KUKA KRL program: p01drop_1711.src, p01drop_1711.dat

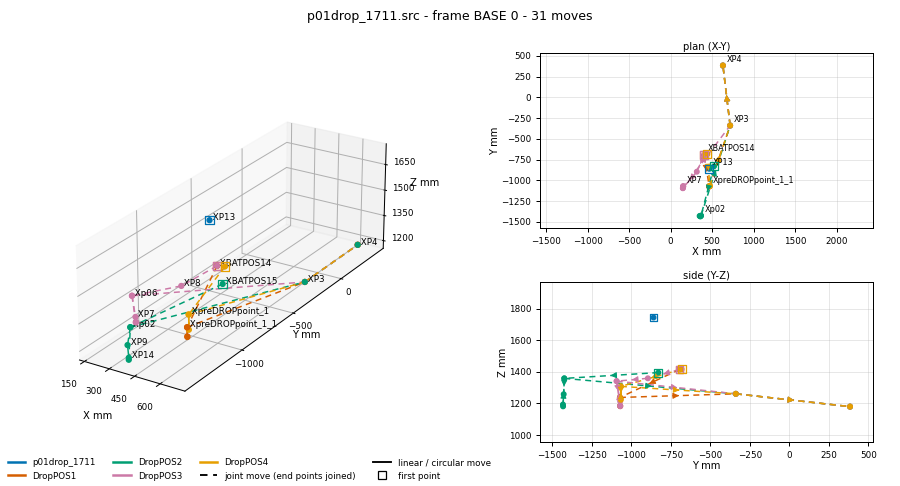
[picture p0: tool path of p01drop_1711.src in frame BASE 0, 31 of 34 moves have a stored position in this frame; points joined in program order, loops and branches not executed]
--- p01drop_1711.src ---
&ACCESS RVP1
&COMMENT Drop Part
&PARAM EDITMASK = *
&PARAM TEMPLATE = C:\KRC\Roboter\Template\vorgabe
&PARAM DISKPATH = KRC:\R1\Program\Sub Programs
DEF p01drop_1711( )
;FOLD INI
  ;FOLD BASISTECH INI

    GLOBAL INTERRUPT DECL 3 WHEN $STOPMESS==TRUE DO IR_STOPM ( )
    INTERRUPT ON 3
    BAS (#INITMOV,0 )
  ;ENDFOLD (BASISTECH INI)
;ENDFOLD (INI)
;================================================
; MODEL    : XXXX
; IE GROUP : XX
; STATION  : XXX
; ROBOT    : RX
; FUNCTION : Drop Part in StXX
;================================================
$TIMER[7]=0
$TIMER_STOP[7]=FALSE

waitarea:
QR_NOK=FALSE

;Wait For Area / Goto Safety / Return To Home

;FOLD PTP P13 Vel=100 % PDAT28 Tool[1] Base[0];%{PE}%R 8.3.48,%MKUKATPBASIS,%CMOVE,%VPTP,%P 1:PTP, 2:P13, 3:, 5:100, 7:PDAT28
$BWDSTART=FALSE
PDAT_ACT=PPDAT28
FDAT_ACT=FP13
BAS(#PTP_PARAMS,100)
PTP XP13
;ENDFOLD
;IF FALSE THEN


WAIT FOR ($IN[54]==TRUE) OR ($IN[1]==TRUE)

IF $in[54]==TRUE THEN
   bomberos_2 ( )               ; PICK In Station XX
   ENDIF


;Para de contar TC hasta que recibe typinfo para dejar (paleta indexada, tipo...)
$TIMER_STOP[7]=TRUE

;FOLD TYPE INFO

WAIT FOR ($IN[54]==TRUE) OR ($IN[1]==TRUE)
IF $in[54]==TRUE THEN
   bomberos_2 ( )               ; PICK In Station XX
   ENDIF
O_TYPE_REQ=FALSE
WAIT FOR I_TYPE_INFO==0
O_TYPE_REQ=TRUE
WAIT FOR ((I_TYPE_INFO>100) AND (I_TYPE_INFO<201) or ($IN[54]==TRUE))
IF $in[54]==TRUE THEN
   bomberos_2 ( )               ; PICK In Station XX
   ENDIF
O_TYPE_INFO=I_TYPE_INFO
;ENDFOLD
;ENDIF

$TIMER_STOP[7]=FALSE

SWITCH i_TYPE_INFO ;coldplate grande o peq


CASE 111
   INDICE_DROP=1 ;Variable calculo TC
   O_TYPE_REQ=FALSE
   DropPOS1() ;POSICION 1 COLDPLATE GRANDE

CASE 112
   INDICE_DROP=2  ;Variable calculo TC
   O_TYPE_REQ=FALSE
   DropPOS2() ;POSICION 2 COLDPLATE GRANDE

CASE 113
   INDICE_DROP=3
   O_TYPE_REQ=FALSE
   DropPOS3() ;POSICION 3 COLDPLATE GRANDE

CASE 121
   INDICE_DROP=4
   O_TYPE_REQ=FALSE
   DropPOS1();POSICION 1 COLDPLATE PEQUEÑO

CASE 200
   INDICE_DROP=4
   O_TYPE_REQ=FALSE
   P01DROP2_2();POSICION 1 COLDPLATE PEQUEÑO

CASE 155
   O_TYPE_REQ=FALSE
   bomberos_2() ;POSICION 1 COLDPLATE GRANDE
DEFAULT

WAIT FOR FALSE

ENDSWITCH

;fold QR NOK
IF (QR_NOK==TRUE) THEN

GOTO waitarea
ENDIF

;ENDFOLD


;FOLD PROVISIONAL PARA PRUEBAS
IF M2_TYPE_INFO<13 THEN
M2_TYPE_INFO=M2_TYPE_INFO+1
ENDIF

;ENDFOLD

PEXIT:

;FOLD Guarda_TC Dejada

;Guarda TC dejada
$TIMER_STOP[7]=TRUE
TC_DROP[INDICE_DROP]=$TIMER[7]

IF (INDICE_DROP < 4) THEN ;CUANDO DEJA ARRAYS EN COLD PLATES GRANDES
   IF (INDICE_RACK == 1)THEN
      TC_CP_BIG[INDICE_DROP]=TC_DROP[INDICE_DROP]+TC_PICK_RACK1[INDICE_PICK]
   ELSE
      TC_CP_BIG[INDICE_DROP]=TC_DROP[INDICE_DROP]+TC_PICK_RACK2[INDICE_PICK]
   ENDIF
   IF (INDICE_DROP == 3) THEN ;Cuando rellena el tercer colplate acumula en array de CP big
      TC_ARRAY_CPB[INDICE_ARRAYS_CPB]=TC_CP_BIG[1]+TC_CP_BIG[2]+TC_CP_BIG[3]
      INDICE_ARRAYS_CPB=INDICE_ARRAYS_CPB+1
      IF (INDICE_ARRAYS_CPB > 18) THEN
         INDICE_ARRAYS_CPB=1
         ;Actualiza el tiempo de ciclo medio por bateria
         ;Toma el tiempo de ciclo medio por batería como la media de procesar 2 racks
         ;64 arrays y 4 cartones, eso vienen a ser unas 7 baterías y me sobra 1 array
         TC_MEDIO_CARTONES=((((TC_CARTON[1]+TC_CARTON[2]+TC_CARTON[3]+TC_CARTON[4])/1000)*63)/64)
         TC_MEDIO_BATERIA=((TC_ARRAY_CPB[1]+TC_ARRAY_CPB[2]+TC_ARRAY_CPB[3]+TC_ARRAY_CPB[4]+TC_ARRAY_CPB[5]+TC_ARRAY_CPB[6]+TC_ARRAY_CPB[7]+TC_ARRAY_CPB[8]+TC_ARRAY_CPB[9]+TC_ARRAY_CPB[10]+TC_ARRAY_CPB[11]+TC_ARRAY_CPB[12]+TC_ARRAY_CPB[13]+TC_ARRAY_CPB[14]+TC_ARRAY_CPB[15]+TC_ARRAY_CPB[16]+TC_ARRAY_CPB[17]+TC_ARRAY_CPB[18]+TC_CP_SMALL[1]+TC_CP_SMALL[2]+TC_CP_SMALL[3]+TC_CP_SMALL[4]+TC_CP_SMALL[5]+TC_CP_SMALL[6]+TC_CP_SMALL[7]+TC_CP_SMALL[8]+TC_CP_SMALL[9])/1000)
         TC_MEDIO_BATERIA=((TC_MEDIO_BATERIA+TC_MEDIO_CARTONES)/9)
      ENDIF
   ENDIF
      ENDIF

IF (INDICE_DROP == 4) THEN ;CUANDO DEJA ARRAYS EN COLD PLATE PEQUEÑOS
   IF (INDICE_RACK == 1)THEN
      TC_CP_SMALL[INDICE_ARRAYS_CPS]=TC_DROP[4]+TC_PICK_RACK1[INDICE_PICK]
   ELSE
      TC_CP_SMALL[INDICE_ARRAYS_CPS]=TC_DROP[4]+TC_PICK_RACK2[INDICE_PICK]
   ENDIF
   INDICE_ARRAYS_CPS=INDICE_ARRAYS_CPS+1
   IF (INDICE_ARRAYS_CPS > 9) THEN
      INDICE_ARRAYS_CPS=1
   ENDIF
ENDIF

;ENDFOLD

END
DEF       DropPOS1()


;FOLD PTP BATPOS14 Vel=100 % PDAT9 Tool[8]:Gripper_array Base[0];%{PE}%R 8.3.48,%MKUKATPBASIS,%CMOVE,%VPTP,%P 1:PTP, 2:BATPOS14, 3:, 5:100, 7:PDAT9
$BWDSTART=FALSE
PDAT_ACT=PPDAT9
FDAT_ACT=FBATPOS14
BAS(#PTP_PARAMS,100)
PTP XBATPOS14
;ENDFOLD
;Wait For Area / Goto Safety / Return To Home

;FOLD Fordtech.Area_Req Area Request: 3, Safety Position: 0, Return To Home: 0 ;%{PE}
Area_Req (3,0,0)
IF I_RETHP AND (0 <> 0) AND ($IN_HOME == TRUE) THEN
  GOTO PEXIT
ENDIF
;ENDFOLD


;FOLD PTP preDROPpoint_1_1 CONT Vel=100 % PDAT9 Tool[8]:Gripper_array Base[0];%{PE}%R 8.3.48,%MKUKATPBASIS,%CMOVE,%VPTP,%P 1:PTP, 2:preDROPpoint_1_1, 3:C_DIS, 5:100, 7:PDAT9
$BWDSTART=FALSE
PDAT_ACT=PPDAT9
FDAT_ACT=FpreDROPpoint_1_1
BAS(#PTP_PARAMS,100)
PTP XpreDROPpoint_1_1 C_DIS
;ENDFOLD

;Pto antes de tocar TIM inclina vert
;FOLD LIN P11 Vel=2 m/s CPDAT9 Tool[8]:Gripper_array Base[0];%{PE}%R 8.3.48,%MKUKATPBASIS,%CMOVE,%VLIN,%P 1:LIN, 2:P11, 3:, 5:2, 7:CPDAT9
$BWDSTART=FALSE
LDAT_ACT=LCPDAT9
FDAT_ACT=FP11
BAS(#CP_PARAMS,2)
LIN XP11
;ENDFOLD
;FOLD WAIT Time=0.3 sec;%{PE}%R 8.3.48,%MKUKATPBASIS,%CWAIT,%VWAIT,%P 3:0.3
WAIT SEC 0.3
;ENDFOLD

;FOLD LIN DROPpoint_1_1 Vel=0.0025 m/s L2 Tool[8]:Gripper_array Base[0];%{PE}%R 8.3.48,%MKUKATPBASIS,%CMOVE,%VLIN,%P 1:LIN, 2:DROPpoint_1_1, 3:, 5:0.0025, 7:L2
$BWDSTART=FALSE
LDAT_ACT=LL2
FDAT_ACT=FDROPpoint_1_1
BAS(#CP_PARAMS,0.0025)
LIN XDROPpoint_1_1
;ENDFOLD

;abrir gara
cil_bat_reposo()

;FOLD PTP preDROPpoint_1_1 CONT Vel=100 % PDAT20 Tool[8]:Gripper_array Base[0];%{PE}%R 8.3.48,%MKUKATPBASIS,%CMOVE,%VPTP,%P 1:PTP, 2:preDROPpoint_1_1, 3:C_DIS, 5:100, 7:PDAT20
$BWDSTART=FALSE
PDAT_ACT=PPDAT20
FDAT_ACT=FpreDROPpoint_1_1
BAS(#PTP_PARAMS,100)
PTP XpreDROPpoint_1_1 C_DIS
;ENDFOLD
;FOLD SYN OUT 43 'Job Ready 3' State=TRUE at START Delay=0 ms;%{PE}%R 8.3.48,%MKUKATPBASIS,%COUT,%VSYNOUT,%P 2:43, 3:Job Ready 3, 5:TRUE, 7:0, 9:0, 12:0
TRIGGER WHEN DISTANCE=0 DELAY=0 DO $OUT[43]=TRUE
;ENDFOLD


;FOLD PTP P3 CONT Vel=100 % PDAT9 Tool[5] Base[0];%{PE}%R 8.3.48,%MKUKATPBASIS,%CMOVE,%VPTP,%P 1:PTP, 2:P3, 3:C_DIS, 5:100, 7:PDAT9
$BWDSTART=FALSE
PDAT_ACT=PPDAT9
FDAT_ACT=FP3
BAS(#PTP_PARAMS,100)
PTP XP3 C_DIS
;ENDFOLD

;Release Area 1
;FOLD SYN OUT 19 'Area Release 3' State=TRUE at START Delay=0 ms;%{PE}%R 8.3.48,%MKUKATPBASIS,%COUT,%VSYNOUT,%P 2:19, 3:Area Release 3, 5:TRUE, 7:0, 9:0, 12:0
TRIGGER WHEN DISTANCE=0 DELAY=0 DO $OUT[19]=TRUE
;ENDFOLD


;FOLD PTP P4 CONT Vel=100 % PDAT9 Tool[5] Base[0];%{PE}%R 8.3.48,%MKUKATPBASIS,%CMOVE,%VPTP,%P 1:PTP, 2:P4, 3:C_DIS, 5:100, 7:PDAT9
$BWDSTART=FALSE
PDAT_ACT=PPDAT9
FDAT_ACT=FP4
BAS(#PTP_PARAMS,100)
PTP XP4 C_DIS
;ENDFOLD

;FOLD PTP HOME Vel=100 % DEFAULT;%{PE}%R 8.3.48,%MKUKATPBASIS,%CMOVE,%VPTP,%P 1:PTP, 2:HOME, 3:, 5:100, 7:DEFAULT
$BWDSTART=FALSE
PDAT_ACT=PDEFAULT
FDAT_ACT=FHOME
BAS(#PTP_PARAMS,100)
$H_POS=XHOME
PTP XHOME
;ENDFOLD
;Jump Adress
PEXIT:



END

DEF       DropPOS2()

;FOLD PTP BATPOS15 Vel=100 % PDAT11 Tool[8]:Gripper_array Base[0];%{PE}%R 8.3.48,%MKUKATPBASIS,%CMOVE,%VPTP,%P 1:PTP, 2:BATPOS15, 3:, 5:100, 7:PDAT11
$BWDSTART=FALSE
PDAT_ACT=PPDAT11
FDAT_ACT=FBATPOS15
BAS(#PTP_PARAMS,100)
PTP XBATPOS15
;ENDFOLD
;Wait For Area / Goto Safety / Return To Home

;FOLD Fordtech.Area_Req Area Request: 3, Safety Position: 0, Return To Home: 0 ;%{PE}
Area_Req (3,0,0)
IF I_RETHP AND (0 <> 0) AND ($IN_HOME == TRUE) THEN
  GOTO PEXIT
ENDIF
;ENDFOLD

;predrop pos
;FOLD PTP p02 CONT Vel=100 % PDAT12 Tool[8]:Gripper_array Base[0];%{PE}%R 8.3.48,%MKUKATPBASIS,%CMOVE,%VPTP,%P 1:PTP, 2:p02, 3:C_DIS, 5:100, 7:PDAT12
$BWDSTART=FALSE
PDAT_ACT=PPDAT12
FDAT_ACT=Fp02
BAS(#PTP_PARAMS,100)
PTP Xp02 C_DIS
;ENDFOLD
;FOLD PTP P9 CONT Vel=100 % PDAT27 Tool[8]:Gripper_array Base[0];%{PE}%R 8.3.48,%MKUKATPBASIS,%CMOVE,%VPTP,%P 1:PTP, 2:P9, 3:C_DIS, 5:100, 7:PDAT27
$BWDSTART=FALSE
PDAT_ACT=PPDAT27
FDAT_ACT=FP9
BAS(#PTP_PARAMS,100)
PTP XP9 C_DIS
;ENDFOLD

;Pto antes de tocar TIM inclina hor
;FOLD LIN P14 Vel=2 m/s CPDAT12 Tool[8]:Gripper_array Base[0];%{PE}%R 8.3.48,%MKUKATPBASIS,%CMOVE,%VLIN,%P 1:LIN, 2:P14, 3:, 5:2, 7:CPDAT12
$BWDSTART=FALSE
LDAT_ACT=LCPDAT12
FDAT_ACT=FP14
BAS(#CP_PARAMS,2)
LIN XP14
;ENDFOLD
;FOLD WAIT Time=0.3 sec;%{PE}%R 8.3.48,%MKUKATPBASIS,%CWAIT,%VWAIT,%P 3:0.3
WAIT SEC 0.3
;ENDFOLD

;drop pos
;FOLD LIN p01 Vel=0.005 m/s L2 Tool[8]:Gripper_array Base[0];%{PE}%R 8.3.48,%MKUKATPBASIS,%CMOVE,%VLIN,%P 1:LIN, 2:p01, 3:, 5:0.005, 7:L2
$BWDSTART=FALSE
LDAT_ACT=LL2
FDAT_ACT=Fp01
BAS(#CP_PARAMS,0.005)
LIN Xp01
;ENDFOLD

;abrir gara
cil_bat_reposo()

;FOLD PTP p02 CONT Vel=100 % PDAT21 Tool[8]:Gripper_array Base[0];%{PE}%R 8.3.48,%MKUKATPBASIS,%CMOVE,%VPTP,%P 1:PTP, 2:p02, 3:C_DIS, 5:100, 7:PDAT21
$BWDSTART=FALSE
PDAT_ACT=PPDAT21
FDAT_ACT=Fp02
BAS(#PTP_PARAMS,100)
PTP Xp02 C_DIS
;ENDFOLD

;FOLD SYN OUT 43 'Job Ready 3' State=TRUE at START Delay=0 ms;%{PE}%R 8.3.48,%MKUKATPBASIS,%COUT,%VSYNOUT,%P 2:43, 3:Job Ready 3, 5:TRUE, 7:0, 9:0, 12:0
TRIGGER WHEN DISTANCE=0 DELAY=0 DO $OUT[43]=TRUE
;ENDFOLD

;FOLD PTP p03 CONT Vel=100 % PDAT13 Tool[5] Base[0];%{PE}%R 8.3.48,%MKUKATPBASIS,%CMOVE,%VPTP,%P 1:PTP, 2:p03, 3:C_DIS, 5:100, 7:PDAT13
$BWDSTART=FALSE
PDAT_ACT=PPDAT13
FDAT_ACT=Fp03
BAS(#PTP_PARAMS,100)
PTP Xp03 C_DIS
;ENDFOLD

;Release Area 1
;FOLD SYN OUT 19 'Area Release 3' State=TRUE at START Delay=0 ms;%{PE}%R 8.3.48,%MKUKATPBASIS,%COUT,%VSYNOUT,%P 2:19, 3:Area Release 3, 5:TRUE, 7:0, 9:0, 12:0
TRIGGER WHEN DISTANCE=0 DELAY=0 DO $OUT[19]=TRUE
;ENDFOLD


;FOLD PTP p04 CONT Vel=100 % PDAT14 Tool[5] Base[0];%{PE}%R 8.3.48,%MKUKATPBASIS,%CMOVE,%VPTP,%P 1:PTP, 2:p04, 3:C_DIS, 5:100, 7:PDAT14
$BWDSTART=FALSE
PDAT_ACT=PPDAT14
FDAT_ACT=Fp04
BAS(#PTP_PARAMS,100)
PTP Xp04 C_DIS
;ENDFOLD

;FOLD PTP HOME Vel=100 % DEFAULT;%{PE}%R 8.3.48,%MKUKATPBASIS,%CMOVE,%VPTP,%P 1:PTP, 2:HOME, 3:, 5:100, 7:DEFAULT
$BWDSTART=FALSE
PDAT_ACT=PDEFAULT
FDAT_ACT=FHOME
BAS(#PTP_PARAMS,100)
$H_POS=XHOME
PTP XHOME
;ENDFOLD
;Jump Adress
PEXIT:

END
DEF       DropPOS3()

;FOLD PTP BATPOS16 Vel=100 % PDAT17 Tool[8]:Gripper_array Base[0];%{PE}%R 8.3.48,%MKUKATPBASIS,%CMOVE,%VPTP,%P 1:PTP, 2:BATPOS16, 3:, 5:100, 7:PDAT17
$BWDSTART=FALSE
PDAT_ACT=PPDAT17
FDAT_ACT=FBATPOS16
BAS(#PTP_PARAMS,100)
PTP XBATPOS16
;ENDFOLD
;Wait For Area / Goto Safety / Return To Home

;FOLD Fordtech.Area_Req Area Request: 3, Safety Position: 0, Return To Home: 0 ;%{PE}
Area_Req (3,0,0)
IF I_RETHP AND (0 <> 0) AND ($IN_HOME == TRUE) THEN
  GOTO PEXIT
ENDIF
;ENDFOLD

;predroppos
;FOLD PTP P8 CONT Vel=100 % PDAT26 Tool[8]:Gripper_array Base[0];%{PE}%R 8.3.48,%MKUKATPBASIS,%CMOVE,%VPTP,%P 1:PTP, 2:P8, 3:C_DIS, 5:100, 7:PDAT26
$BWDSTART=FALSE
PDAT_ACT=PPDAT26
FDAT_ACT=FP8
BAS(#PTP_PARAMS,100)
PTP XP8 C_DIS
;ENDFOLD
;FOLD PTP p06 CONT Vel=100 % PDAT16 Tool[8]:Gripper_array Base[0];%{PE}%R 8.3.48,%MKUKATPBASIS,%CMOVE,%VPTP,%P 1:PTP, 2:p06, 3:C_DIS, 5:100, 7:PDAT16
$BWDSTART=FALSE
PDAT_ACT=PPDAT16
FDAT_ACT=Fp06
BAS(#PTP_PARAMS,100)
PTP Xp06 C_DIS
;ENDFOLD
;FOLD PTP P7 CONT Vel=100 % PDAT25 Tool[8]:Gripper_array Base[0];%{PE}%R 8.3.48,%MKUKATPBASIS,%CMOVE,%VPTP,%P 1:PTP, 2:P7, 3:C_DIS, 5:100, 7:PDAT25
$BWDSTART=FALSE
PDAT_ACT=PPDAT25
FDAT_ACT=FP7
BAS(#PTP_PARAMS,100)
PTP XP7 C_DIS
;ENDFOLD

;Pto antes de tocar TIM
;FOLD LIN P12 Vel=2 m/s CPDAT11 Tool[8]:Gripper_array Base[0];%{PE}%R 8.3.48,%MKUKATPBASIS,%CMOVE,%VLIN,%P 1:LIN, 2:P12, 3:, 5:2, 7:CPDAT11
$BWDSTART=FALSE
LDAT_ACT=LCPDAT11
FDAT_ACT=FP12
BAS(#CP_PARAMS,2)
LIN XP12
;ENDFOLD
;FOLD WAIT Time=0.3 sec;%{PE}%R 8.3.48,%MKUKATPBASIS,%CWAIT,%VWAIT,%P 3:0.3
WAIT SEC 0.3
;ENDFOLD

;droppos
;FOLD LIN p05 Vel=0.0025 m/s L2 Tool[8]:Gripper_array Base[0];%{PE}%R 8.3.48,%MKUKATPBASIS,%CMOVE,%VLIN,%P 1:LIN, 2:p05, 3:, 5:0.0025, 7:L2
$BWDSTART=FALSE
LDAT_ACT=LL2
FDAT_ACT=Fp05
BAS(#CP_PARAMS,0.0025)
LIN Xp05
;ENDFOLD

;abrir gara
cil_bat_reposo()

;FOLD PTP p06 CONT Vel=100 % PDAT22 Tool[8]:Gripper_array Base[0];%{PE}%R 8.3.48,%MKUKATPBASIS,%CMOVE,%VPTP,%P 1:PTP, 2:p06, 3:C_DIS, 5:100, 7:PDAT22
$BWDSTART=FALSE
PDAT_ACT=PPDAT22
FDAT_ACT=Fp06
BAS(#PTP_PARAMS,100)
PTP Xp06 C_DIS
;ENDFOLD


;FOLD SYN OUT 43 'Job Ready 3' State=TRUE at START Delay=0 ms;%{PE}%R 8.3.48,%MKUKATPBASIS,%COUT,%VSYNOUT,%P 2:43, 3:Job Ready 3, 5:TRUE, 7:0, 9:0, 12:0
TRIGGER WHEN DISTANCE=0 DELAY=0 DO $OUT[43]=TRUE
;ENDFOLD

;FOLD PTP p07 CONT Vel=100 % PDAT18 Tool[5] Base[0];%{PE}%R 8.3.48,%MKUKATPBASIS,%CMOVE,%VPTP,%P 1:PTP, 2:p07, 3:C_DIS, 5:100, 7:PDAT18
$BWDSTART=FALSE
PDAT_ACT=PPDAT18
FDAT_ACT=Fp07
BAS(#PTP_PARAMS,100)
PTP Xp07 C_DIS
;ENDFOLD

;Release Area 1
;FOLD SYN OUT 19 'Area Release 3' State=TRUE at START Delay=0 ms;%{PE}%R 8.3.48,%MKUKATPBASIS,%COUT,%VSYNOUT,%P 2:19, 3:Area Release 3, 5:TRUE, 7:0, 9:0, 12:0
TRIGGER WHEN DISTANCE=0 DELAY=0 DO $OUT[19]=TRUE
;ENDFOLD


;FOLD PTP p08 CONT Vel=100 % PDAT19 Tool[5] Base[0];%{PE}%R 8.3.48,%MKUKATPBASIS,%CMOVE,%VPTP,%P 1:PTP, 2:p08, 3:C_DIS, 5:100, 7:PDAT19
$BWDSTART=FALSE
PDAT_ACT=PPDAT19
FDAT_ACT=Fp08
BAS(#PTP_PARAMS,100)
PTP Xp08 C_DIS
;ENDFOLD

;FOLD PTP HOME Vel=100 % DEFAULT;%{PE}%R 8.3.48,%MKUKATPBASIS,%CMOVE,%VPTP,%P 1:PTP, 2:HOME, 3:, 5:100, 7:DEFAULT
$BWDSTART=FALSE
PDAT_ACT=PDEFAULT
FDAT_ACT=FHOME
BAS(#PTP_PARAMS,100)
$H_POS=XHOME
PTP XHOME
;ENDFOLD
;Jump Adress
PEXIT:



END
DEF       DropPOS4()

;FOLD PTP BATPOS13 Vel=100 % PDAT8 Tool[5] Base[0];%{PE}%R 8.3.48,%MKUKATPBASIS,%CMOVE,%VPTP,%P 1:PTP, 2:BATPOS13, 3:, 5:100, 7:PDAT8
$BWDSTART=FALSE
PDAT_ACT=PPDAT8
FDAT_ACT=FBATPOS13
BAS(#PTP_PARAMS,100)
PTP XBATPOS13
;ENDFOLD
;Wait For Area / Goto Safety / Return To Home

;FOLD Fordtech.Area_Req Area Request: 3, Safety Position: 0, Return To Home: 0 ;%{PE}
Area_Req (3,0,0)
IF I_RETHP AND (0 <> 0) AND ($IN_HOME == TRUE) THEN
  GOTO PEXIT
ENDIF
;ENDFOLD

;FOLD PTP preDROPpoint_1 CONT Vel=100 % PDAT8 Tool[5] Base[0];%{PE}%R 8.3.48,%MKUKATPBASIS,%CMOVE,%VPTP,%P 1:PTP, 2:preDROPpoint_1, 3:C_DIS, 5:100, 7:PDAT8
$BWDSTART=FALSE
PDAT_ACT=PPDAT8
FDAT_ACT=FpreDROPpoint_1
BAS(#PTP_PARAMS,100)
PTP XpreDROPpoint_1 C_DIS
;ENDFOLD

;FOLD LIN DROPpoint_1 Vel=0.5 m/s L Tool[5]:Gripper_empty Base[0];%{PE}%R 8.3.48,%MKUKATPBASIS,%CMOVE,%VLIN,%P 1:LIN, 2:DROPpoint_1, 3:, 5:0.5, 7:L
$BWDSTART=FALSE
LDAT_ACT=LL
FDAT_ACT=FDROPpoint_1
BAS(#CP_PARAMS,0.5)
LIN XDROPpoint_1
;ENDFOLD

;abrir gara
cil_bat_reposo()

;FOLD LIN preDROPpoint_1 Vel=2 m/s CPDAT4 Tool[5] Base[0];%{PE}%R 8.3.48,%MKUKATPBASIS,%CMOVE,%VLIN,%P 1:LIN, 2:preDROPpoint_1, 3:, 5:2, 7:CPDAT4
$BWDSTART=FALSE
LDAT_ACT=LCPDAT4
FDAT_ACT=FpreDROPpoint_1
BAS(#CP_PARAMS,2)
LIN XpreDROPpoint_1
;ENDFOLD
;FOLD Fordtech.Job_Rdy Set Job Ready: 3   ;%{PE}
Job_Ready (3)
;ENDFOLD


;FOLD PTP P1 CONT Vel=100 % PDAT8 Tool[5] Base[0];%{PE}%R 8.3.48,%MKUKATPBASIS,%CMOVE,%VPTP,%P 1:PTP, 2:P1, 3:C_DIS, 5:100, 7:PDAT8
$BWDSTART=FALSE
PDAT_ACT=PPDAT8
FDAT_ACT=FP1
BAS(#PTP_PARAMS,100)
PTP XP1 C_DIS
;ENDFOLD
;FOLD PTP P2 CONT Vel=100 % PDAT8 Tool[5] Base[0];%{PE}%R 8.3.48,%MKUKATPBASIS,%CMOVE,%VPTP,%P 1:PTP, 2:P2, 3:C_DIS, 5:100, 7:PDAT8
$BWDSTART=FALSE
PDAT_ACT=PPDAT8
FDAT_ACT=FP2
BAS(#PTP_PARAMS,100)
PTP XP2 C_DIS
;ENDFOLD

;Release Area 1
;FOLD Fordtech.Area_Rel Area Release: 3   ;%{PE}
Area_Rel (3)
;ENDFOLD

;Jump Adress
PEXIT:




END

--- p01drop_1711.dat ---
&ACCESS RVP1
&COMMENT Drop Part
&PARAM EDITMASK = *
&PARAM TEMPLATE = C:\KRC\Roboter\Template\vorgabe
&PARAM DISKPATH = KRC:\R1\Program\Sub Programs
DEFDAT p01drop_1711

EXT  BAS (BAS_COMMAND  :IN,REAL  :IN )
DECL INT SUCCESS
;******************************
;*     E6POS Declarations     *
;******************************

DECL E6POS XP01WAITREQ2={X 2157.35596,Y -301.755188,Z 2852.14893,A -15.8183,B 72.8074417,C -9.82211304,S 2,T 34,E1 0.0,E2 0.0,E3 0.0,E4 0.0,E5 0.0,E6 0.0}
DECL E6POS XP10={X 2411.43896,Y 1748.73096,Z -1095.62903,A -177.692307,B -16.9195194,C 42.7874298,S 2,T 34,E1 0.0,E2 0.0,E3 0.0,E4 0.0,E5 0.0,E6 0.0}
DECL E6POS XP20={X 1670.59900,Y -157.831207,Z 2354.64209,A -15.8183,B 72.8074417,C -9.82211304,S 2,T 34,E1 0.0,E2 0.0,E3 0.0,E4 0.0,E5 0.0,E6 0.0}
DECL E6POS XP30={X 1670.59900,Y -157.831207,Z 2354.64209,A -15.8183,B 72.8074417,C -9.82211304,S 2,T 34,E1 0.0,E2 0.0,E3 0.0,E4 0.0,E5 0.0,E6 0.0}
DECL E6POS XDROP_POS={X 1670.59900,Y -157.831207,Z 2354.64209,A -15.8183,B 72.8074417,C -9.82211304,S 2,T 34,E1 0.0,E2 0.0,E3 0.0,E4 0.0,E5 0.0,E6 0.0}
DECL E6POS XP40={X 2411.43896,Y 1748.73096,Z -1095.62903,A -177.692307,B -16.9195194,C 42.7874298,S 2,T 34,E1 0.0,E2 0.0,E3 0.0,E4 0.0,E5 0.0,E6 0.0}
DECL E6POS XP50={X 2411.43896,Y 1748.73096,Z -1095.62903,A -177.692307,B -16.9195194,C 42.7874298,S 2,T 34,E1 0.0,E2 0.0,E3 0.0,E4 0.0,E5 0.0,E6 0.0}
DECL E6POS XP01WAITREL2={X 2411.43896,Y 1748.73096,Z -1095.62903,A -177.692307,B -16.9195194,C 42.7874298,S 2,T 34,E1 0.0,E2 0.0,E3 0.0,E4 0.0,E5 0.0,E6 0.0}

;******************************
;*     FDAT Declarations      *
;******************************

DECL FDAT FP01WAITREQ2={TOOL_NO 12,BASE_NO 0,IPO_FRAME #BASE}
DECL FDAT FP10={TOOL_NO 12,BASE_NO 0,IPO_FRAME #TCP}
DECL FDAT FP20={TOOL_NO 12,BASE_NO 0,IPO_FRAME #TCP}
DECL FDAT FP30={TOOL_NO 12,BASE_NO 0,IPO_FRAME #TCP}
DECL FDAT FDROP_POS={TOOL_NO 12,BASE_NO 0,IPO_FRAME #TCP}
DECL FDAT FP40={TOOL_NO 12,BASE_NO 0,IPO_FRAME #TCP}
DECL FDAT FP50={TOOL_NO 12,BASE_NO 0,IPO_FRAME #TCP}
DECL FDAT FP01WAITREL2={TOOL_NO 12,BASE_NO 0,IPO_FRAME #TCP}

;******************************
;*  PDAT & LDAT Declarations  *
;******************************

DECL PDAT PH={VEL 100.000,ACC 100.000,APO_DIST 100.000,APO_MODE #CDIS,GEAR_JERK 100.000,EXAX_IGN 0}

DECL MODULEPARAM_T LAST_TP_PARAMS={PARAMS[] "FORDTECH.P_AREA_REQ=3; FORDTECH.P_SAFETY_POS=0; FORDTECH.P_RET=0; Kuka.VelocityFieldEnabled=False; Kuka.ColDetectFieldEnabled=False; Kuka.MovementParameterFieldEnabled=False; Kuka.IsAngleEnabled=False; Kuka.PointName=P01Waitdrop; Kuka.FrameData.base_no=0; Kuka.FrameData.tool_no=12; Kuka.FrameData.ipo_frame=#BASE; Kuka.isglobalpoint=False; Kuka.MoveDataPtpName=H; Kuka.MovementDataPdat.apo_mode=#CDIS; Kuka.MovementDataPdat.apo_dist=100; Kuka.MovementData.vel=100; Kuka.MovementData.acc=100; Kuka.MovementData.exax_ign=0; Kuka.VelocityPtp=100; Kuka.BlendingEnabled=False; Kuka.APXEnabled=False; Kuka.CurrentCDSetIndex=0"}
DECL E6POS XP01Waitdrop={X 290.951508,Y 816.177185,Z 1155.55042,A -86.9976196,B 22.0779018,C -179.006119,S 6,T 27,E1 0.0,E2 0.0,E3 0.0,E4 0.0,E5 0.0,E6 0.0}
DECL FDAT FP01Waitdrop={TOOL_NO 5,BASE_NO 0,IPO_FRAME #BASE,POINT2[] " ",TQ_STATE FALSE}
DECL BASIS_SUGG_T LAST_BASIS={POINT1[] "P0                      ",POINT2[] "P0                      ",CP_PARAMS[] "CPDAT0                  ",PTP_PARAMS[] "PDAT0                   ",CONT[] "                        ",CP_VEL[] "0.005                   ",PTP_VEL[] "100                     ",SYNC_PARAMS[] "SYNCDAT                 ",SPL_NAME[] "S0                      ",A_PARAMS[] "ADAT0                   "}
DECL E6POS XP1WAITDROP={X -1019.53088,Y 1662.02295,Z 1494.18030,A -87.0150070,B 22.0766544,C -179.006226,S 6,T 27,E1 0.0,E2 0.0,E3 0.0,E4 0.0,E5 0.0,E6 0.0}
DECL FDAT FP1Waitdrop={TOOL_NO 12,BASE_NO 0,IPO_FRAME #BASE,POINT2[] " ",TQ_STATE FALSE}
DECL PDAT PPDAT1={VEL 100.000,ACC 100.000,APO_DIST 100.000,GEAR_JERK 50.0000,EXAX_IGN 0}
DECL E6POS XP2WAITDROP={X 442.124359,Y -682.465210,Z 1416.05603,A -171.206314,B 14.8656197,C -154.747955,S 6,T 26,E1 0.0,E2 0.0,E3 0.0,E4 0.0,E5 0.0,E6 0.0}
DECL FDAT FP2Waitdrop={TOOL_NO 8,BASE_NO 0,IPO_FRAME #BASE,POINT2[] " ",TQ_STATE FALSE}
DECL PDAT PPDAT2={VEL 100.000,ACC 100.000,APO_DIST 100.000,GEAR_JERK 50.0000,EXAX_IGN 0}
DECL E6POS XP03drop_1={X 1357.71619,Y -332.386230,Z 1270.87256,A 92.5587387,B 7.42240524,C 175.886597,S 6,T 26,E1 0.0,E2 0.0,E3 0.0,E4 0.0,E5 0.0,E6 0.0}
DECL FDAT FP03drop_1={TOOL_NO 12,BASE_NO 0,IPO_FRAME #BASE,POINT2[] " ",TQ_STATE FALSE}
DECL PDAT PPDAT4={VEL 100.000,ACC 100.000,APO_DIST 100.000,GEAR_JERK 50.0000,EXAX_IGN 0}
DECL E6POS XP02drop_1={X 1435.38062,Y -451.789185,Z 1034.59302,A 89.9487686,B 4.10017967,C -172.489868,S 6,T 26,E1 0.0,E2 0.0,E3 0.0,E4 0.0,E5 0.0,E6 0.0}
DECL FDAT FP02drop_1={TOOL_NO 12,BASE_NO 0,IPO_FRAME #BASE,POINT2[] " ",TQ_STATE FALSE}
DECL PDAT PPDAT3={VEL 100.000,ACC 100.000,APO_DIST 100.000,GEAR_JERK 50.0000,EXAX_IGN 0}
DECL E6POS XP2={X 629.440857,Y 383.904541,Z 1179.93518,A -112.750427,B 20.1261520,C -170.604736,S 6,T 27,E1 0.0,E2 0.0,E3 0.0,E4 0.0,E5 0.0,E6 0.0}
DECL FDAT FP2={TOOL_NO 5,BASE_NO 0,IPO_FRAME #BASE,POINT2[] " ",TQ_STATE FALSE}
DECL PDAT PPDAT8={VEL 100.000,ACC 100.000,APO_DIST 100.000,APO_MODE #CDIS,GEAR_JERK 50.0000,EXAX_IGN 0}
DECL E6POS XP1={X 716.539490,Y -339.002350,Z 1261.05945,A -151.411957,B 9.54572201,C -170.760315,S 6,T 26,E1 0.0,E2 0.0,E3 0.0,E4 0.0,E5 0.0,E6 0.0}
DECL FDAT FP1={TOOL_NO 5,BASE_NO 0,IPO_FRAME #BASE,POINT2[] " ",TQ_STATE FALSE}
DECL PDAT PPDAT7={VEL 100.000,ACC 100.000,APO_DIST 100.000,APO_MODE #CDIS,GEAR_JERK 50.0000,EXAX_IGN 0}
DECL LDAT LCPDAT4={VEL 2.00000,ACC 100.000,APO_DIST 100.000,APO_FAC 50.0000,AXIS_VEL 100.000,AXIS_ACC 100.000,ORI_TYP #VAR,CIRC_TYP #BASE,JERK_FAC 50.0000,GEAR_JERK 50.0000,EXAX_IGN 0}
DECL E6POS XDROPpoint_1={X 471.147,Y -1067.04773,Z 1223.22400,A -179.451859,B -0.162765205,C 179.769058,S 6,T 26,E1 0.0,E2 0.0,E3 0.0,E4 0.0,E5 0.0,E6 0.0}
DECL FDAT FDROPpoint_1={TOOL_NO 5,BASE_NO 0,IPO_FRAME #BASE,POINT2[] " ",TQ_STATE FALSE}
DECL LDAT LCPDAT3={VEL 2.00000,ACC 100.000,APO_DIST 100.000,APO_FAC 50.0000,AXIS_VEL 100.000,AXIS_ACC 100.000,ORI_TYP #VAR,CIRC_TYP #BASE,JERK_FAC 50.0000,GEAR_JERK 50.0000,EXAX_IGN 0}
DECL E6POS XpreDROPpoint_1={X 471.147,Y -1067.04773,Z 1308.08960,A -179.451859,B -0.162765205,C 179.769058,S 6,T 26,E1 0.0,E2 0.0,E3 0.0,E4 0.0,E5 0.0,E6 0.0}
DECL FDAT FpreDROPpoint_1={TOOL_NO 5,BASE_NO 0,IPO_FRAME #BASE,POINT2[] " ",TQ_STATE FALSE}
DECL PDAT PPDAT6={VEL 100.000,ACC 100.000,APO_DIST 100.000,APO_MODE #CDIS,GEAR_JERK 50.0000,EXAX_IGN 0}
DECL E6POS XBATPOS13={X 442.124359,Y -682.465210,Z 1416.05603,A -171.206314,B 14.8656197,C -154.747955,S 6,T 26,E1 0.0,E2 0.0,E3 0.0,E4 0.0,E5 0.0,E6 0.0}
DECL FDAT FBATPOS13={TOOL_NO 5,BASE_NO 0,IPO_FRAME #BASE,POINT2[] " ",TQ_STATE FALSE}
DECL PDAT PPDAT5={VEL 100.000,ACC 100.000,APO_DIST 100.000,GEAR_JERK 50.0000,EXAX_IGN 0}
DECL E6POS XP4={X 629.440857,Y 383.904541,Z 1179.93518,A -112.750427,B 20.1261520,C -170.604736,S 6,T 27,E1 0.0,E2 0.0,E3 0.0,E4 0.0,E5 0.0,E6 0.0}
DECL FDAT FP4={TOOL_NO 5,BASE_NO 0,IPO_FRAME #BASE,POINT2[] " ",TQ_STATE FALSE}
DECL E6POS XP3={X 716.539490,Y -339.002350,Z 1261.05945,A -151.411957,B 9.54572201,C -170.760315,S 6,T 26,E1 0.0,E2 0.0,E3 0.0,E4 0.0,E5 0.0,E6 0.0}
DECL FDAT FP3={TOOL_NO 5,BASE_NO 0,IPO_FRAME #BASE,POINT2[] " ",TQ_STATE FALSE}
DECL LDAT LCPDAT6={VEL 2.00000,ACC 100.000,APO_DIST 100.000,APO_FAC 50.0000,AXIS_VEL 100.000,AXIS_ACC 100.000,ORI_TYP #VAR,CIRC_TYP #BASE,JERK_FAC 50.0000,GEAR_JERK 50.0000,EXAX_IGN 0}
DECL E6POS XDROPpoint_1_1={X 464.376862,Y -1070.86938,Z 1182.52637,A -179.823196,B -0.162590399,C 179.884659,S 6,T 26,E1 0.0,E2 0.0,E3 0.0,E4 0.0,E5 0.0,E6 0.0}
DECL FDAT FDROPpoint_1_1={TOOL_NO 8,BASE_NO 0,IPO_FRAME #BASE,POINT2[] " ",TQ_STATE FALSE}
DECL LDAT LCPDAT5={VEL 2.00000,ACC 100.000,APO_DIST 100.000,APO_FAC 50.0000,AXIS_VEL 100.000,AXIS_ACC 100.000,ORI_TYP #VAR,CIRC_TYP #BASE,JERK_FAC 50.0000,GEAR_JERK 50.0000,EXAX_IGN 0}
DECL E6POS XpreDROPpoint_1_1={X 464.811249,Y -1073.00403,Z 1237.95544,A -179.724121,B -0.162587121,C -179.891113,S 6,T 26,E1 0.0,E2 0.0,E3 0.0,E4 0.0,E5 0.0,E6 0.0}
DECL FDAT FpreDROPpoint_1_1={TOOL_NO 8,BASE_NO 0,IPO_FRAME #BASE,POINT2[] " ",TQ_STATE FALSE}
DECL E6POS XBATPOS14={X 403.061340,Y -695.623413,Z 1415.04932,A -162.936142,B 2.48320770,C -179.431671,S 6,T 26,E1 0.0,E2 0.0,E3 0.0,E4 0.0,E5 0.0,E6 0.0}
DECL FDAT FBATPOS14={TOOL_NO 8,BASE_NO 0,IPO_FRAME #BASE,POINT2[] " ",TQ_STATE FALSE}
DECL PDAT PPDAT9={VEL 100.000,ACC 100.000,APO_DIST 100.000,APO_MODE #CDIS,GEAR_JERK 50.0000,EXAX_IGN 0}
DECL E6POS XP01={X 357.196228,Y -1432.68530,Z 1181.60425,A 0.145591095,B -0.0267589036,C 179.917831,S 6,T 26,E1 0.0,E2 0.0,E3 0.0,E4 0.0,E5 0.0,E6 0.0}
DECL FDAT Fp01={TOOL_NO 8,BASE_NO 0,IPO_FRAME #BASE,POINT2[] " ",TQ_STATE FALSE}
DECL PDAT PPDAT10={VEL 100.000,ACC 100.000,APO_DIST 100.000,GEAR_JERK 50.0000,EXAX_IGN 0}
DECL LDAT LCPDAT1={VEL 2.00000,ACC 100.000,APO_DIST 100.000,APO_FAC 50.0000,AXIS_VEL 100.000,AXIS_ACC 100.000,ORI_TYP #VAR,CIRC_TYP #BASE,JERK_FAC 50.0000,GEAR_JERK 50.0000,EXAX_IGN 0}
DECL PDAT PPDAT11={VEL 100.000,ACC 100.000,APO_DIST 100.000,APO_MODE #CDIS,GEAR_JERK 50.0000,EXAX_IGN 0}
DECL E6POS XBATPOS15={X 522.221252,Y -830.045410,Z 1395.37085,A 178.482819,B 10.0271606,C -166.759811,S 6,T 26,E1 0.0,E2 0.0,E3 0.0,E4 0.0,E5 0.0,E6 0.0}
DECL FDAT FBATPOS15={TOOL_NO 8,BASE_NO 0,IPO_FRAME #BASE,POINT2[] " ",TQ_STATE FALSE}
DECL E6POS XP02={X 365.452240,Y -1425.07288,Z 1358.66589,A 0.347011298,B 0.208950698,C -179.836838,S 6,T 26,E1 0.0,E2 0.0,E3 0.0,E4 0.0,E5 0.0,E6 0.0}
DECL FDAT Fp02={TOOL_NO 8,BASE_NO 0,IPO_FRAME #BASE,POINT2[] " ",TQ_STATE FALSE}
DECL PDAT PPDAT12={VEL 100.000,ACC 100.000,APO_DIST 100.000,APO_MODE #CDIS,GEAR_JERK 50.0000,EXAX_IGN 0}
DECL LDAT LCPDAT2={VEL 2.00000,ACC 100.000,APO_DIST 100.000,APO_FAC 50.0000,AXIS_VEL 100.000,AXIS_ACC 100.000,ORI_TYP #VAR,CIRC_TYP #BASE,JERK_FAC 50.0000,GEAR_JERK 50.0000,EXAX_IGN 0}
DECL PDAT PPDAT13={VEL 100.000,ACC 100.000,APO_DIST 100.000,APO_MODE #CDIS,GEAR_JERK 50.0000,EXAX_IGN 0}
DECL E6POS Xp03={X 716.539490,Y -339.002350,Z 1261.05945,A -151.411957,B 9.54572201,C -170.760315,S 6,T 26,E1 0.0,E2 0.0,E3 0.0,E4 0.0,E5 0.0,E6 0.0}
DECL FDAT Fp03={TOOL_NO 5,BASE_NO 0,IPO_FRAME #BASE,POINT2[] " ",TQ_STATE FALSE}
DECL PDAT PPDAT14={VEL 100.000,ACC 100.000,APO_DIST 100.000,APO_MODE #CDIS,GEAR_JERK 50.0000,EXAX_IGN 0}
DECL E6POS Xp04={X 629.440857,Y 383.904541,Z 1179.93518,A -112.750427,B 20.1261520,C -170.604736,S 6,T 27,E1 0.0,E2 0.0,E3 0.0,E4 0.0,E5 0.0,E6 0.0}
DECL FDAT Fp04={TOOL_NO 5,BASE_NO 0,IPO_FRAME #BASE,POINT2[] " ",TQ_STATE FALSE}
DECL E6POS XP05={X 150.799423,Y -1070.86938,Z 1182.78,A -179.823196,B -0.162590489,C 179.884659,S 6,T 26,E1 0.0,E2 0.0,E3 0.0,E4 0.0,E5 0.0,E6 0.0}
DECL FDAT Fp05={TOOL_NO 8,BASE_NO 0,IPO_FRAME #BASE,POINT2[] " ",TQ_STATE FALSE}
DECL PDAT PPDAT15={VEL 100.000,ACC 100.000,APO_DIST 100.000,APO_MODE #CDIS,GEAR_JERK 50.0000,EXAX_IGN 0}
DECL E6POS XP06={X 146.841568,Y -1093.77332,Z 1341.20703,A 179.704926,B -11.1497049,C -178.051468,S 6,T 26,E1 0.0,E2 0.0,E3 0.0,E4 0.0,E5 0.0,E6 0.0}
DECL FDAT Fp06={TOOL_NO 8,BASE_NO 0,IPO_FRAME #BASE,POINT2[] " ",TQ_STATE FALSE}
DECL PDAT PPDAT16={VEL 100.000,ACC 100.000,APO_DIST 100.000,APO_MODE #CDIS,GEAR_JERK 50.0000,EXAX_IGN 0}
DECL PDAT PPDAT17={VEL 100.000,ACC 100.000,APO_DIST 100.000,APO_MODE #CDIS,GEAR_JERK 50.0000,EXAX_IGN 0}
DECL E6POS XBATPOS16={X 403.061340,Y -695.623413,Z 1415.04932,A -162.936142,B 2.48320770,C -179.431671,S 6,T 26,E1 0.0,E2 0.0,E3 0.0,E4 0.0,E5 0.0,E6 0.0}
DECL FDAT FBATPOS16={TOOL_NO 8,BASE_NO 0,IPO_FRAME #BASE,POINT2[] " ",TQ_STATE FALSE}
DECL LDAT LCPDAT7={VEL 2.00000,ACC 100.000,APO_DIST 100.000,APO_FAC 50.0000,AXIS_VEL 100.000,AXIS_ACC 100.000,ORI_TYP #VAR,CIRC_TYP #BASE,JERK_FAC 50.0000,GEAR_JERK 50.0000,EXAX_IGN 0}
DECL PDAT PPDAT18={VEL 100.000,ACC 100.000,APO_DIST 100.000,APO_MODE #CDIS,GEAR_JERK 50.0000,EXAX_IGN 0}
DECL E6POS Xp07={X 716.539490,Y -339.002350,Z 1261.05945,A -151.411957,B 9.54572201,C -170.760315,S 6,T 26,E1 0.0,E2 0.0,E3 0.0,E4 0.0,E5 0.0,E6 0.0}
DECL FDAT Fp07={TOOL_NO 5,BASE_NO 0,IPO_FRAME #BASE,POINT2[] " ",TQ_STATE FALSE}
DECL PDAT PPDAT19={VEL 100.000,ACC 100.000,APO_DIST 100.000,APO_MODE #CDIS,GEAR_JERK 50.0000,EXAX_IGN 0}
DECL E6POS Xp08={X 629.440857,Y 383.904541,Z 1179.93518,A -112.750427,B 20.1261520,C -170.604736,S 6,T 27,E1 0.0,E2 0.0,E3 0.0,E4 0.0,E5 0.0,E6 0.0}
DECL FDAT Fp08={TOOL_NO 5,BASE_NO 0,IPO_FRAME #BASE,POINT2[] " ",TQ_STATE FALSE}
DECL LDAT LCPDAT8={VEL 2.00000,ACC 100.000,APO_DIST 100.000,APO_FAC 50.0000,AXIS_VEL 100.000,AXIS_ACC 100.000,ORI_TYP #VAR,CIRC_TYP #BASE,JERK_FAC 50.0000,GEAR_JERK 50.0000,EXAX_IGN 0}
DECL PDAT PPDAT20={VEL 100.000,ACC 100.000,APO_DIST 100.000,APO_MODE #CDIS,GEAR_JERK 50.0000,EXAX_IGN 0}
DECL PDAT PPDAT21={VEL 100.000,ACC 100.000,APO_DIST 100.000,APO_MODE #CDIS,GEAR_JERK 50.0000,EXAX_IGN 0}
DECL PDAT PPDAT22={VEL 100.000,ACC 100.000,APO_DIST 100.000,APO_MODE #CDIS,GEAR_JERK 50.0000,EXAX_IGN 0}
DECL E6POS XP5={X 464.811249,Y -1073.00403,Z 1237.95544,A -179.724121,B -0.162587121,C -179.891113,S 6,T 26,E1 0.0,E2 0.0,E3 0.0,E4 0.0,E5 0.0,E6 0.0}
DECL FDAT FP5={TOOL_NO 8,BASE_NO 0,IPO_FRAME #BASE,POINT2[] " ",TQ_STATE FALSE}
DECL PDAT PPDAT23={VEL 100.000,ACC 100.000,APO_DIST 100.000,APO_MODE #CDIS,GEAR_JERK 50.0000,EXAX_IGN 0}
DECL E6POS XP6={X 358.421143,Y -1434.49048,Z 1213.64075,A 0.238015085,B -0.0266249236,C 179.917816,S 6,T 26,E1 0.0,E2 0.0,E3 0.0,E4 0.0,E5 0.0,E6 0.0}
DECL FDAT FP6={TOOL_NO 8,BASE_NO 0,IPO_FRAME #BASE,POINT2[] " ",TQ_STATE FALSE}
DECL PDAT PPDAT24={VEL 100.000,ACC 100.000,APO_DIST 100.000,APO_MODE #CDIS,GEAR_JERK 50.0000,EXAX_IGN 0}
DECL E6POS XP7={X 150.063629,Y -1071.55493,Z 1214.23828,A 179.805801,B -0.441522,C 179.922180,S 6,T 26,E1 0.0,E2 0.0,E3 0.0,E4 0.0,E5 0.0,E6 0.0}
DECL FDAT FP7={TOOL_NO 8,BASE_NO 0,IPO_FRAME #BASE,POINT2[] " ",TQ_STATE FALSE}
DECL PDAT PPDAT25={VEL 100.000,ACC 100.000,APO_DIST 100.000,APO_MODE #CDIS,GEAR_JERK 50.0000,EXAX_IGN 0}
DECL E6POS XP8={X 314.908356,Y -895.846313,Z 1359.21680,A -177.333069,B 1.31368983,C -165.688553,S 6,T 26,E1 0.0,E2 0.0,E3 0.0,E4 0.0,E5 0.0,E6 0.0}
DECL FDAT FP8={TOOL_NO 8,BASE_NO 0,IPO_FRAME #BASE,POINT2[] " ",TQ_STATE FALSE}
DECL PDAT PPDAT26={VEL 100.000,ACC 100.000,APO_DIST 100.000,APO_MODE #CDIS,GEAR_JERK 50.0000,EXAX_IGN 0}
DECL E6POS XP9={X 349.023438,Y -1428.75208,Z 1258.37793,A 0.251577318,B 0.00656803325,C 179.944351,S 6,T 26,E1 0.0,E2 0.0,E3 0.0,E4 0.0,E5 0.0,E6 0.0}
DECL FDAT FP9={TOOL_NO 8,BASE_NO 0,IPO_FRAME #BASE,POINT2[] " ",TQ_STATE FALSE}
DECL PDAT PPDAT27={VEL 100.000,ACC 100.000,APO_DIST 100.000,APO_MODE #CDIS,GEAR_JERK 50.0000,EXAX_IGN 0}
DECL E6POS XP11={X 464.368439,Y -1071.24353,Z 1186.03467,A -179.823196,B -0.162590399,C -179.316956,S 6,T 26,E1 0.0,E2 0.0,E3 0.0,E4 0.0,E5 0.0,E6 0.0}
DECL FDAT FP11={TOOL_NO 8,BASE_NO 0,IPO_FRAME #BASE,POINT2[] " ",TQ_STATE FALSE}
DECL LDAT LCPDAT9={VEL 2.00000,ACC 100.000,APO_DIST 100.000,APO_FAC 50.0000,AXIS_VEL 100.000,AXIS_ACC 100.000,ORI_TYP #VAR,CIRC_TYP #BASE,JERK_FAC 50.0000,GEAR_JERK 50.0000,EXAX_IGN 0}
DECL LDAT LCPDAT10={VEL 2.00000,ACC 100.000,APO_DIST 100.000,APO_FAC 50.0000,AXIS_VEL 100.000,AXIS_ACC 100.000,ORI_TYP #VAR,CIRC_TYP #BASE,JERK_FAC 50.0000,GEAR_JERK 50.0000,EXAX_IGN 0}
DECL E6POS XP12={X 151.782639,Y -1071.24353,Z 1186.03467,A -179.823196,B -0.162590429,C -179.316956,S 6,T 26,E1 0.0,E2 0.0,E3 0.0,E4 0.0,E5 0.0,E6 0.0}
DECL FDAT FP12={TOOL_NO 8,BASE_NO 0,IPO_FRAME #BASE,POINT2[] " ",TQ_STATE FALSE}
DECL LDAT LCPDAT11={VEL 2.00000,ACC 100.000,APO_DIST 100.000,APO_FAC 50.0000,AXIS_VEL 100.000,AXIS_ACC 100.000,ORI_TYP #VAR,CIRC_TYP #BASE,JERK_FAC 50.0000,GEAR_JERK 50.0000,EXAX_IGN 0}
DECL E6POS XP13={X 464.934357,Y -860.178223,Z 1744.02759,A -162.936142,B 2.48320770,C -179.431671,S 6,T 26,E1 0.0,E2 0.0,E3 0.0,E4 0.0,E5 0.0,E6 0.0}
DECL FDAT FP13={TOOL_NO 1,BASE_NO 0,IPO_FRAME #BASE,POINT2[] " ",TQ_STATE FALSE}
DECL PDAT PPDAT28={VEL 100.000,ACC 100.000,APO_DIST 100.000,GEAR_JERK 50.0000,EXAX_IGN 0}
DECL LDAT LL={VEL 2.00000,ACC 25.0000,APO_DIST 100.000,APO_FAC 50.0000,AXIS_VEL 100.000,AXIS_ACC 100.000,ORI_TYP #VAR,CIRC_TYP #BASE,JERK_FAC 50.0000,GEAR_JERK 50.0000,EXAX_IGN 0}
DECL E6POS XP14={X 358.055664,Y -1433.38574,Z 1193.16907,A 0.408299953,B -0.0297936238,C 178.499512,S 6,T 26,E1 0.0,E2 0.0,E3 0.0,E4 0.0,E5 0.0,E6 0.0}
DECL FDAT FP14={TOOL_NO 8,BASE_NO 0,IPO_FRAME #BASE,POINT2[] " ",TQ_STATE FALSE}
DECL LDAT LCPDAT12={VEL 2.00000,ACC 100.000,APO_DIST 100.000,APO_FAC 50.0000,AXIS_VEL 100.000,AXIS_ACC 100.000,ORI_TYP #VAR,CIRC_TYP #BASE,JERK_FAC 50.0000,GEAR_JERK 50.0000,EXAX_IGN 0}
DECL LDAT LL2={VEL 2.00000,ACC 10.0000,APO_DIST 100.000,APO_FAC 50.0000,AXIS_VEL 100.000,AXIS_ACC 100.000,ORI_TYP #VAR,CIRC_TYP #BASE,JERK_FAC 50.0000,GEAR_JERK 50.0000,EXAX_IGN 0}
ENDDAT
